(*

.. <legal notes>

legal notes
=================
| SPDX-FileCopyrightText: © 2026 Oleksandr Tiutyk <trofimich@gmail.com>
| SPDX-License-Identifier: LGPL-3.0-only
| For details check: LGPL-3.0-only_

.. _LGPL-3.0-only: https://www.gnu.org/licenses/lgpl-3.0.en.html

.. </legal notes>

*)

FUNCTION_BLOCK ABSTRACT SimpleDevice EXTENDS Device

PROPERTY PROTECTED FINAL InternalChildCount : Core.INT_INDEX
GET
InternalChildCount := 0;
END_GET
END_PROPERTY

METHOD PROTECTED InternalTryGetChildByIndex : IChildAutomationComponent
VAR_INPUT
	index : Core.INT_INDEX;
END_VAR
InternalTryGetChildByIndex := 0;
END_METHOD

END_FUNCTION_BLOCK

(* stored: Version 1.1.0.1
   POU SimpleDevice: Id {7c21300f-1ad4-4217-9d49-d0f060249ecb}, SpecialFunc None
   Folder Overriden members: Id {185562e6-4d51-4174-9462-636590f15fda}
   Property InternalChildCount: Id {2fd0f5c0-dd77-4f98-b857-5fe55eabb827}
   Get Get: Id {291f62b5-aa6f-4982-aecf-8050bd9a9e61}
   Method InternalTryGetChildByIndex: Id {20c59d36-ccf0-4a7d-bcde-dac491881353} *)
